INTERFACE I_LinkedListItem EXTENDS I_LinkedListItem

PROPERTY PUBLIC DataType : T_MaxString
GET
END_GET
END_PROPERTY

METHOD PUBLIC Destroy
VAR_INPUT
END_VAR
END_METHOD

METHOD PUBLIC Equals : BOOL
VAR_INPUT
	Symbol : ANY;
END_VAR
END_METHOD

METHOD PUBLIC Get : BOOL;
VAR_INPUT
	Destination : ANY;
END_VAR
END_METHOD

PROPERTY PUBLIC Next : I_LinkedListItem
GET
END_GET
SET
END_SET
END_PROPERTY

PROPERTY PUBLIC Previous : I_LinkedListItem
GET
END_GET
SET
END_SET
END_PROPERTY

END_INTERFACE

(* stored: Version 1.1.0.1, ProductVersion 3.1.4024.12
   Itf I_LinkedListItem: Id {0cff8fbe-58e6-42f0-93b9-bcbf9ae1547a}
   Property DataType: Id {67a6de58-0b51-42eb-b8e3-c204779e535c}
   Get Get: Id {25cb2f4f-c892-49f2-8386-16628d6fc9b5}
   Method Destroy: Id {63a4bd84-b6d5-48f0-b124-677ef16e8f2b}
   Method Equals: Id {42524c8e-5be9-4ec1-9fd9-53150bfb09c1}
   Method Get: Id {3cf610bf-474c-45ea-8852-ef97d7e3e565}
   Property Next: Id {36f7d60e-da19-4ec7-aef7-5f62014911e7}
   Get Get: Id {e871223f-e76e-40e1-ac6e-8232b4f33a89}
   Set Set: Id {01642d6e-14c4-4289-a99f-8469c57d0bae}
   Property Previous: Id {391f15bb-7210-4ad5-9151-9a7de912f823}
   Get Get: Id {855706cd-3426-4a83-93fc-01ff73e63b41}
   Set Set: Id {d562e515-c3b0-4344-956f-865d275d909b} *)
